{attribute 'GeneratedUsingTerminal: EL5002-0000-0020'}
{attribute addProperty BoxType "EL5002-0000-0020"}
{attribute addProperty Id "EtcSlaveTerminalBaseSSI_Inputs_Channel_1AT %I*SSI_Inputs_Channel_EDA1628411SSI_Inputs_Channel_2AT %I*SSI_Inputs_Channel_EDA1628411WcStateAT %I*WcState_9091E0EB2InfoDataAT %I*InfoData_32EB74EA10"}
{attribute addProperty CRC "3710112345"}
{attribute addProperty Size "34"}
TYPE EL5002_DD23D259 EXTENDS EtcSlaveTerminalBase :
STRUCT
	{attribute addProperty Name "SSI_Inputs_Channel_1"}
	SSI_Inputs_Channel_1 : SSI_Inputs_Channel_EDA16284;
	{attribute addProperty Name "SSI_Inputs_Channel_2"}
	SSI_Inputs_Channel_2 : SSI_Inputs_Channel_EDA16284;
	{attribute addProperty Name "WcState"}
	WcState : WcState_9091E0EB;
	{attribute addProperty Name "InfoData"}
	InfoData : InfoData_32EB74EA;
END_STRUCT
END_TYPE

(* stored: Version 1.2.0.0, ProductVersion 3.1.4024.9
   DUT EL5002_DD23D259: Id {106a683a-88ca-42a6-8ed0-f7ece6675fa8} *)
